// Mitsubishi GX Works2 project: BookEX6_7 Time   PLC: Q13UDV

// global labels: Global
VAR_GLOBAL
  bVar0 AT M5000 : BOOL;
  abArray0 AT M5010 : ARRAY [0..49] OF BOOL;
  sStr0 AT D5000 : STRING[199];
  sStr1 AT D5100 : STRING[199];
  sStr2 AT D5200 : STRING[199];
  sStr3 AT D5300 : STRING[199];
  sStr4 AT D5400 : STRING[199];
  sStr5 AT D5500 : STRING[199];
  sStr6 AT D5600 : STRING[199];
  sStr7 AT D5700 : STRING[199];
  sStr8 AT D5800 : STRING[199];
  sStr9 AT D5900 : STRING[199];
  iVar0 AT D4500 : INT;
  iVar1 AT D4501 : INT;
  iVar2 AT D4502 : INT;
  iVar3 AT D4503 : INT;
  iVar4 AT D4504 : INT;
  iVar5 AT D4505 : INT;
  iVar6 AT D4506 : INT;
  iVar7 AT D4507 : INT;
  iVar8 AT D4508 : INT;
  iVar9 AT D4509 : INT;
  dVar0 AT D4510 : DINT;
  dVar1 AT D4512 : DINT;
  dVar2 AT D4514 : DINT;
  dVar3 AT D4516 : DINT;
  dVar4 AT D4518 : DINT;
  dVar5 AT D4520 : DINT;
  dVar6 AT D4522 : DINT;
  dVar7 AT D4524 : DINT;
  dVar8 AT D4526 : DINT;
  dVar9 AT D4528 : DINT;
  wVar0 AT D4530 : WORD;
  wVar1 AT D4531 : WORD;
  wVar2 AT D4532 : WORD;
  wVar3 AT D4533 : WORD;
  wVar4 AT D4534 : WORD;
  wVar5 AT D4535 : WORD;
  wVar6 AT D4536 : WORD;
  wVar7 AT D4537 : WORD;
  wVar8 AT D4538 : WORD;
  wVar9 AT D4539 : WORD;
  dwVar0 AT D4540 : DWORD;
  dwVar1 AT D4542 : DWORD;
  dwVar2 AT D4544 : DWORD;
  dwVar3 AT D4546 : DWORD;
  dwVar4 AT D4548 : DWORD;
  dwVar5 AT D4550 : DWORD;
  dwVar6 AT D4552 : DWORD;
  dwVar7 AT D4554 : DWORD;
  dwVar8 AT D4556 : DWORD;
  dwVar9 AT D4558 : DWORD;
  fsVar0 AT D4560 : REAL;
  fsVar1 AT D4562 : REAL;
  fsVar2 AT D4564 : REAL;
  fsVar3 AT D4566 : REAL;
  fsVar4 AT D4568 : REAL;
  fsVar5 AT D4570 : REAL;
  fsVar6 AT D4572 : REAL;
  fsVar7 AT D4574 : REAL;
  fsVar8 AT D4576 : REAL;
  fsVar9 AT D4578 : REAL;
  fdVar0 AT D4580 : LREAL;
  tTime0 AT D4620 : TIME;
  tTime1 AT D4622 : TIME;
  tTime2 AT D4624 : TIME;
  tTime3 AT D4626 : TIME;
  tTime4 AT D4628 : TIME;
  tTime5 AT D4630 : TIME;
  tTime6 AT D4632 : TIME;
  tTime7 AT D4634 : TIME;
  tTime8 AT D4636 : TIME;
  tTime9 AT D4638 : TIME;
  tTime10 AT D4640 : TIME;
  bVar1 AT M5001 : BOOL;
  bVar2 AT M5002 : BOOL;
  bVar3 AT M5003 : BOOL;
  bVar4 AT M5004 : BOOL;
  bVar5 AT M5005 : BOOL;
  bVar6 AT M5006 : BOOL;
  bVar7 AT M5007 : BOOL;
  bVar8 AT M5008 : BOOL;
  bVar9 AT M5009 : BOOL;
  abArray1 AT M5060 : ARRAY [0..49] OF BOOL;
  abArray2 AT M5110 : ARRAY [0..49] OF BOOL;
  abArray3 AT M5160 : ARRAY [0..49] OF BOOL;
  abArray4 AT M5210 : ARRAY [0..49] OF BOOL;
  abArray5 AT M5260 : ARRAY [0..49] OF BOOL;
  abArray6 AT M5310 : ARRAY [0..49] OF BOOL;
  abArray7 AT M5360 : ARRAY [0..49] OF BOOL;
  abArray8 AT M5410 : ARRAY [0..49] OF BOOL;
  abArray9 AT M5460 : ARRAY [0..49] OF BOOL;
  fdVar1 AT D4584 : LREAL;
  fdVar2 AT D4588 : LREAL;
  fdVar3 AT D4592 : LREAL;
  fdVar4 AT D4596 : LREAL;
  fdVar5 AT D4600 : LREAL;
  fdVar6 AT D4604 : LREAL;
  fdVar7 AT D4608 : LREAL;
  fdVar8 AT D4612 : LREAL;
  fdVar9 AT D4616 : LREAL;
END_VAR
// user libraries (not included): HMI

FUNCTION ABS_TIME
VAR_INPUT
  t_IN1 : TIME;
  t_IN2 : TIME;
END_VAR
VAR
  tTemp : TIME;
END_VAR
;
tTemp := SUB_TIME(t_IN1, t_IN2);
IF tTemp < T#0ms THEN
	tTemp := MUL_TIME(tTemp, -1);
END_IF;
ABS_TIME := tTemp;
END_FUNCTION

FUNCTION Day2Time
VAR_INPUT
  fs_IN : REAL;
END_VAR
;
Day2Time := DINT_TO_TIME(REAL_TO_DINT(fs_IN * 86400000.0));
END_FUNCTION

FUNCTION fsDIV_TIME
VAR_INPUT
  t_IN1 : TIME;
  fs_IN2 : REAL;
END_VAR
VAR
  dTemp : DINT;
  fsTemp : REAL;
END_VAR
;
dTemp := TIME_TO_DINT(t_IN1);
fsTemp := DINT_TO_REAL(dTemp) / fs_IN2;
fsDIV_TIME := DINT_TO_TIME(REAL_TO_DINT(fsTemp));
END_FUNCTION

FUNCTION fsMUL_TIME
VAR_INPUT
  t_IN1 : TIME;
  fs_IN2 : REAL;
END_VAR
VAR
  dTemp : DINT;
  fsTemp : REAL;
END_VAR
;
dTemp := TIME_TO_DINT(t_IN1);
fsTemp := DINT_TO_REAL(dTemp) * fs_IN2;
fsMUL_TIME := DINT_TO_TIME(REAL_TO_DINT(fsTemp));
END_FUNCTION

FUNCTION Hour2Time
VAR_INPUT
  fs_IN : REAL;
END_VAR
;
Hour2Time := DINT_TO_TIME(REAL_TO_DINT(fs_IN * 3600000.0));
END_FUNCTION

FUNCTION Min2Time
VAR_INPUT
  fs_IN : REAL;
END_VAR
;
Min2Time := DINT_TO_TIME(REAL_TO_DINT(fs_IN * 60000.0));
END_FUNCTION

FUNCTION Sec2Time
VAR_INPUT
  fs_IN : REAL;
END_VAR
;
Sec2Time := DINT_TO_TIME(REAL_TO_DINT(fs_IN * 1000.0));
END_FUNCTION

PROGRAM ExADDTIME
(* structured ladder/FBD written out as ST: instructions are called as NAME(EN, inputs, outputs); _pN, _eN, _tN stand for wires *)
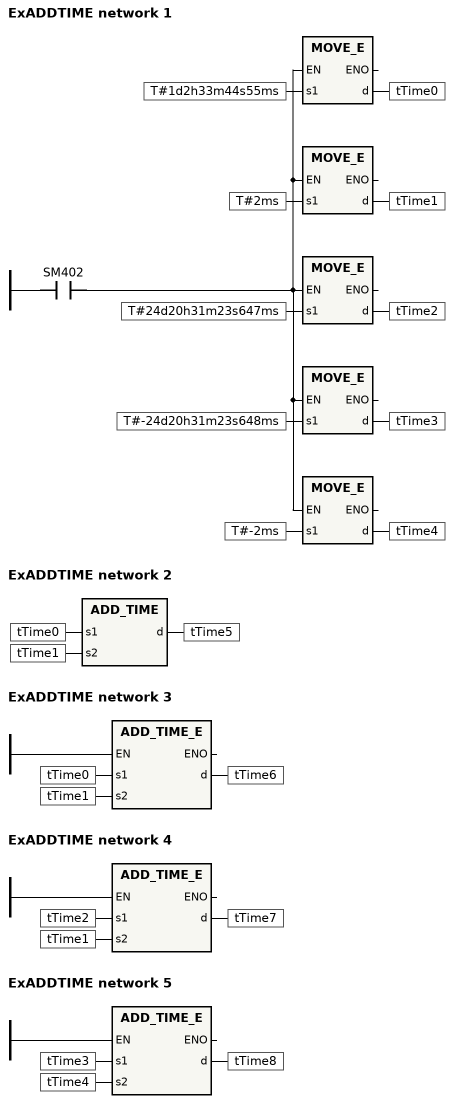
(* network 1 *)
MOVE_E(SM402, T#1d2h33m44s55ms, tTime0);
MOVE_E(SM402, T#2ms, tTime1);
MOVE_E(SM402, T#24d20h31m23s647ms, tTime2);
MOVE_E(SM402, T#-24d20h31m23s648ms, tTime3);
MOVE_E(SM402, T#-2ms, tTime4);
(* network 2 *)
tTime5 := ADD_TIME(tTime0, tTime1);
(* network 3 *)
ADD_TIME_E(TRUE, tTime0, tTime1, tTime6);
(* network 4 *)
ADD_TIME_E(TRUE, tTime2, tTime1, tTime7);
(* network 5 *)
ADD_TIME_E(TRUE, tTime3, tTime4, tTime8);
END_PROGRAM

PROGRAM ExDIVTIME
VAR
  tTime20 : TIME;
  tTime21 : TIME;
  tTime22 : TIME;
  tTime23 : TIME;
  tTime24 : TIME;
  tTime25 : TIME;
  tTime26 : TIME;
  tTime27 : TIME;
  tTime28 : TIME;
  tTime29 : TIME;
END_VAR
(* structured ladder/FBD written out as ST: instructions are called as NAME(EN, inputs, outputs); _pN, _eN, _tN stand for wires *)
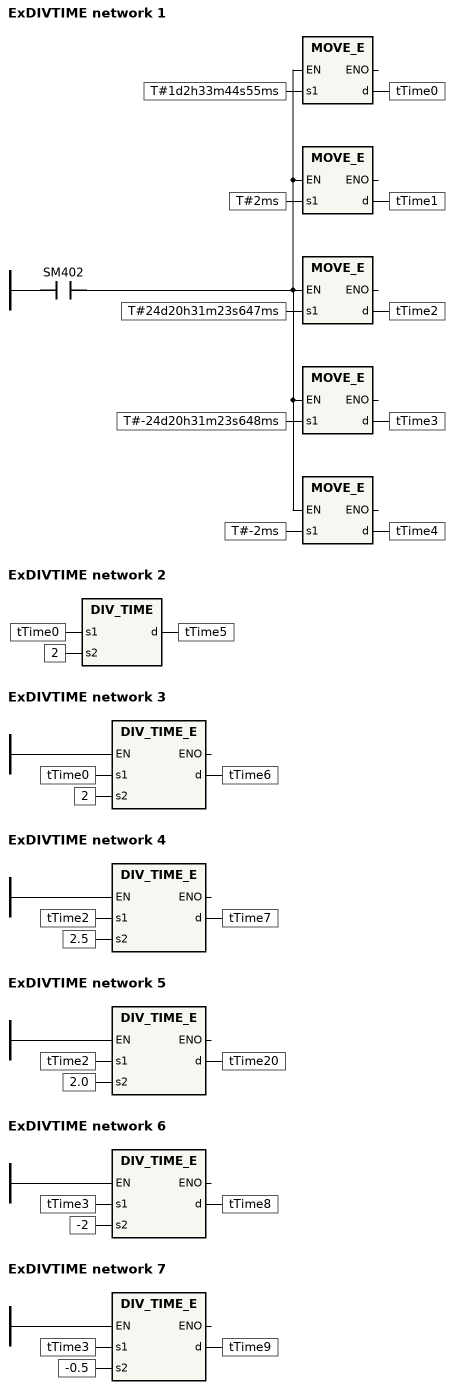
(* network 1 *)
MOVE_E(SM402, T#1d2h33m44s55ms, tTime0);
MOVE_E(SM402, T#2ms, tTime1);
MOVE_E(SM402, T#24d20h31m23s647ms, tTime2);
MOVE_E(SM402, T#-24d20h31m23s648ms, tTime3);
MOVE_E(SM402, T#-2ms, tTime4);
(* network 2 *)
tTime5 := DIV_TIME(tTime0, 2);
(* network 3 *)
DIV_TIME_E(TRUE, tTime0, 2, tTime6);
(* network 4 *)
DIV_TIME_E(TRUE, tTime2, 2.5, tTime7);
(* network 5 *)
DIV_TIME_E(TRUE, tTime2, 2.0, tTime20);
(* network 6 *)
DIV_TIME_E(TRUE, tTime3, -2, tTime8);
(* network 7 *)
DIV_TIME_E(TRUE, tTime3, -0.5, tTime9);
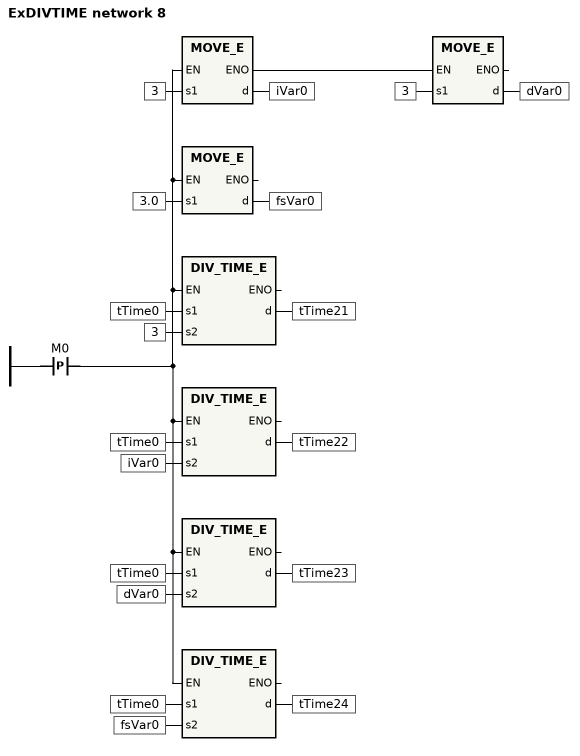
(* network 8 *)
_p1 := LDP(TRUE, M0);
_e2 := MOVE_E(_p1, 3, iVar0);
MOVE_E(_e2, 3, dVar0);
MOVE_E(_p1, 3.0, fsVar0);
DIV_TIME_E(_p1, tTime0, 3, tTime21);
DIV_TIME_E(_p1, tTime0, iVar0, tTime22);
DIV_TIME_E(_p1, tTime0, dVar0, tTime23);
DIV_TIME_E(_p1, tTime0, fsVar0, tTime24);
END_PROGRAM

PROGRAM ExFB
(* structured ladder/FBD written out as ST: instructions are called as NAME(EN, inputs, outputs); _pN, _eN, _tN stand for wires *)
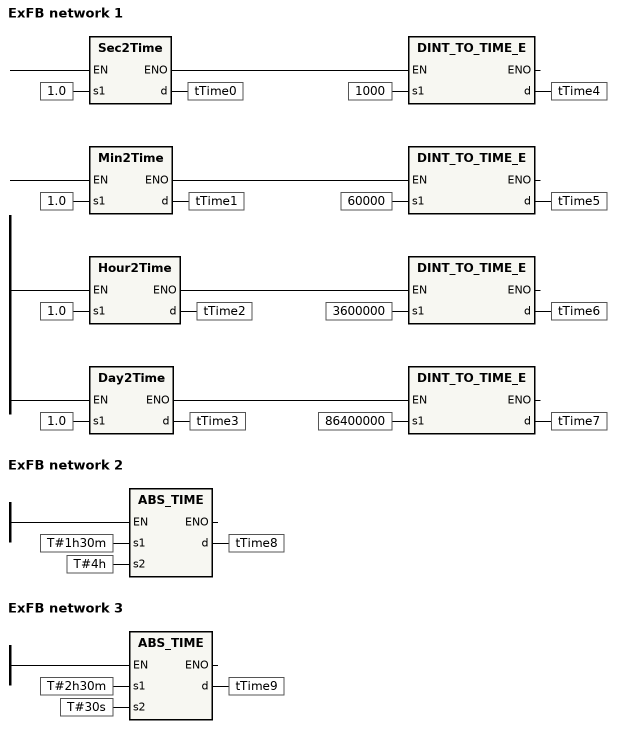
(* network 1 *)
_e1 := Sec2Time(TRUE, 1.0, tTime0);
DINT_TO_TIME_E(_e1, 1000, tTime4);
_e2 := Min2Time(TRUE, 1.0, tTime1);
DINT_TO_TIME_E(_e2, 60000, tTime5);
_e3 := Hour2Time(TRUE, 1.0, tTime2);
DINT_TO_TIME_E(_e3, 3600000, tTime6);
_e4 := Day2Time(TRUE, 1.0, tTime3);
DINT_TO_TIME_E(_e4, 86400000, tTime7);
(* network 2 *)
ABS_TIME(TRUE, T#1h30m, T#4h, tTime8);
(* network 3 *)
ABS_TIME(TRUE, T#2h30m, T#30s, tTime9);
END_PROGRAM

PROGRAM ExMUL_DIV
VAR
  tTime20 : TIME;
  tTime21 : TIME;
  tTime22 : TIME;
  tTime23 : TIME;
  tTime24 : TIME;
  tTime25 : TIME;
  tTime26 : TIME;
  tTime27 : TIME;
  tTime28 : TIME;
  tTime29 : TIME;
  tTime30 : TIME;
  tTime31 : TIME;
  tTime32 : TIME;
  tTime33 : TIME;
  tTime34 : TIME;
  tTime35 : TIME;
  tTime36 : TIME;
  tTime37 : TIME;
  tTime38 : TIME;
  tTime39 : TIME;
  tTime40 : TIME;
END_VAR
(* structured ladder/FBD written out as ST: instructions are called as NAME(EN, inputs, outputs); _pN, _eN, _tN stand for wires *)
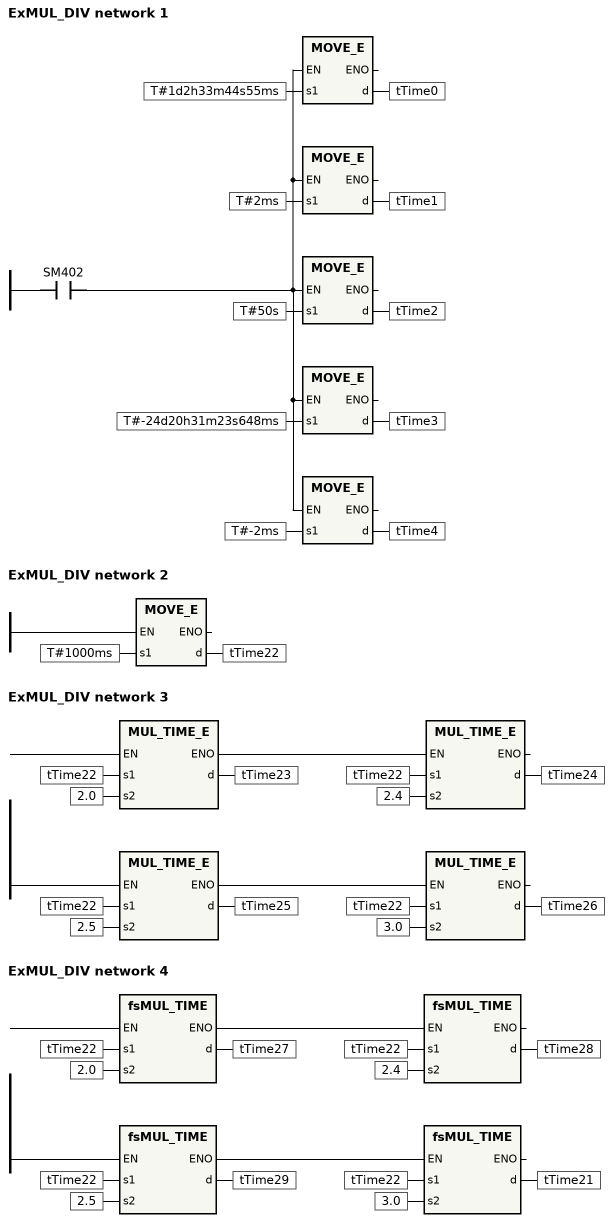
(* network 1 *)
MOVE_E(SM402, T#1d2h33m44s55ms, tTime0);
MOVE_E(SM402, T#2ms, tTime1);
MOVE_E(SM402, T#50s, tTime2);
MOVE_E(SM402, T#-24d20h31m23s648ms, tTime3);
MOVE_E(SM402, T#-2ms, tTime4);
(* network 2 *)
MOVE_E(TRUE, T#1000ms, tTime22);
(* network 3 *)
_e1 := MUL_TIME_E(TRUE, tTime22, 2.0, tTime23);
MUL_TIME_E(_e1, tTime22, 2.4, tTime24);
_e2 := MUL_TIME_E(TRUE, tTime22, 2.5, tTime25);
MUL_TIME_E(_e2, tTime22, 3.0, tTime26);
(* network 4 *)
_e1 := fsMUL_TIME(TRUE, tTime22, 2.0, tTime27);
fsMUL_TIME(_e1, tTime22, 2.4, tTime28);
_e2 := fsMUL_TIME(TRUE, tTime22, 2.5, tTime29);
fsMUL_TIME(_e2, tTime22, 3.0, tTime21);
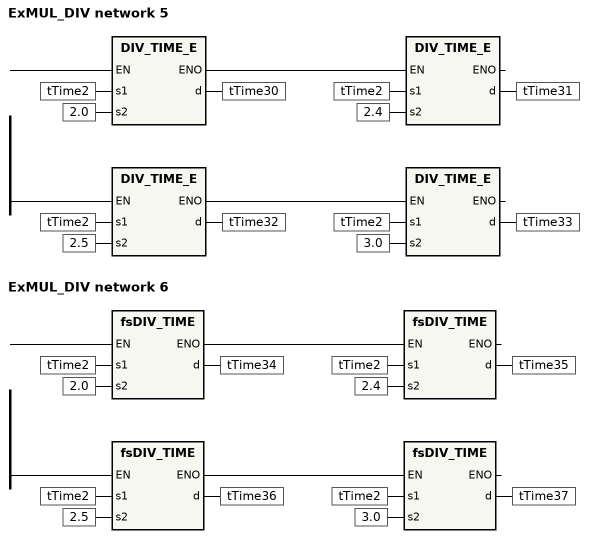
(* network 5 *)
_e1 := DIV_TIME_E(TRUE, tTime2, 2.0, tTime30);
DIV_TIME_E(_e1, tTime2, 2.4, tTime31);
_e2 := DIV_TIME_E(TRUE, tTime2, 2.5, tTime32);
DIV_TIME_E(_e2, tTime2, 3.0, tTime33);
(* network 6 *)
_e1 := fsDIV_TIME(TRUE, tTime2, 2.0, tTime34);
fsDIV_TIME(_e1, tTime2, 2.4, tTime35);
_e2 := fsDIV_TIME(TRUE, tTime2, 2.5, tTime36);
fsDIV_TIME(_e2, tTime2, 3.0, tTime37);
END_PROGRAM

PROGRAM ExMULTIME
(* structured ladder/FBD written out as ST: instructions are called as NAME(EN, inputs, outputs); _pN, _eN, _tN stand for wires *)
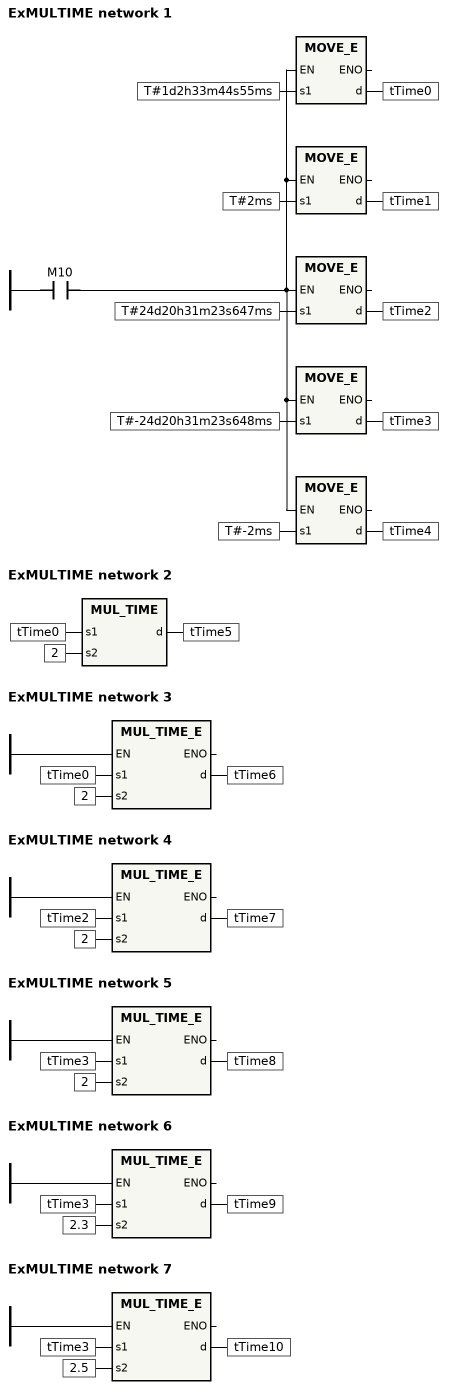
(* network 1 *)
MOVE_E(M10, T#1d2h33m44s55ms, tTime0);
MOVE_E(M10, T#2ms, tTime1);
MOVE_E(M10, T#24d20h31m23s647ms, tTime2);
MOVE_E(M10, T#-24d20h31m23s648ms, tTime3);
MOVE_E(M10, T#-2ms, tTime4);
(* network 2 *)
tTime5 := MUL_TIME(tTime0, 2);
(* network 3 *)
MUL_TIME_E(TRUE, tTime0, 2, tTime6);
(* network 4 *)
MUL_TIME_E(TRUE, tTime2, 2, tTime7);
(* network 5 *)
MUL_TIME_E(TRUE, tTime3, 2, tTime8);
(* network 6 *)
MUL_TIME_E(TRUE, tTime3, 2.3, tTime9);
(* network 7 *)
MUL_TIME_E(TRUE, tTime3, 2.5, tTime10);
END_PROGRAM

PROGRAM ExSUBTIME
(* structured ladder/FBD written out as ST: instructions are called as NAME(EN, inputs, outputs); _pN, _eN, _tN stand for wires *)
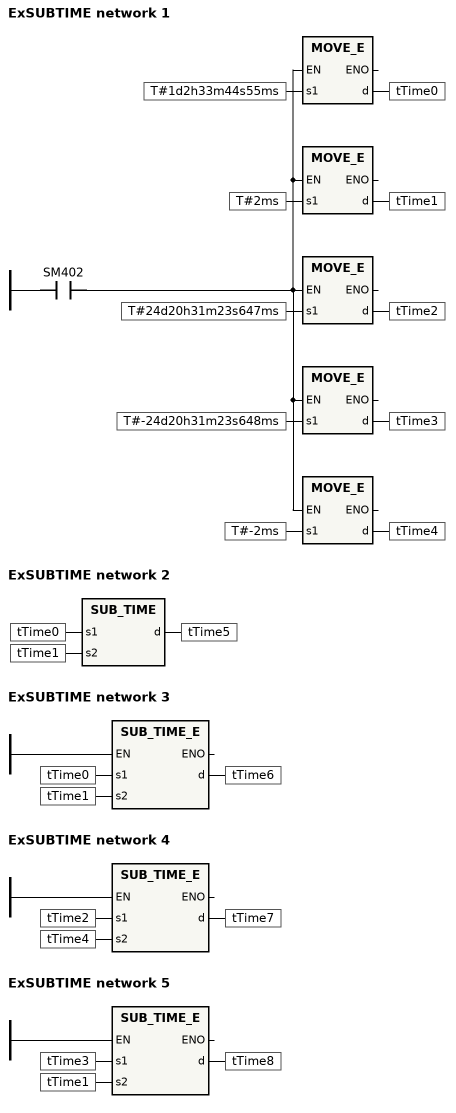
(* network 1 *)
MOVE_E(SM402, T#1d2h33m44s55ms, tTime0);
MOVE_E(SM402, T#2ms, tTime1);
MOVE_E(SM402, T#24d20h31m23s647ms, tTime2);
MOVE_E(SM402, T#-24d20h31m23s648ms, tTime3);
MOVE_E(SM402, T#-2ms, tTime4);
(* network 2 *)
tTime5 := SUB_TIME(tTime0, tTime1);
(* network 3 *)
SUB_TIME_E(TRUE, tTime0, tTime1, tTime6);
(* network 4 *)
SUB_TIME_E(TRUE, tTime2, tTime4, tTime7);
(* network 5 *)
SUB_TIME_E(TRUE, tTime3, tTime1, tTime8);
END_PROGRAM

PROGRAM stt
;
tTime2 := ADD_TIME( tTime0 , tTime1 );
bVar0 := ADD_TIME_E( TRUE,  tTime0 , tTime1, tTime2 );
tTime2 := SUB_TIME( tTime0 , tTime1 );
END_PROGRAM

PROGRAM ExDIV_ST
VAR
  tTime20 : TIME;
  tTime21 : TIME;
  tTime22 : TIME;
  tTime23 : TIME;
  tTime24 : TIME;
  tTime25 : TIME;
  tTime26 : TIME;
  tTime27 : TIME;
  tTime28 : TIME;
  tTime29 : TIME;
  tTime30 : TIME;
  tTime31 : TIME;
  tTime32 : TIME;
  tTime33 : TIME;
  tTime34 : TIME;
  tTime35 : TIME;
  tTime36 : TIME;
  tTime37 : TIME;
  tTime38 : TIME;
  tTime39 : TIME;
END_VAR
;
iVar1 := 3;
dVar1 := 3;
fsVar1 := 3.0;
tTime0 := T#1d2h33m44s55ms;
 
tTime29 := tTime0 + tTime1;
tTime28 := tTime0 - tTime1;

tTime31 := tTime0 * 3;
tTime32 := tTime0 * iVar1;
tTime33 := tTime0 * dVar1;
tTime34 := tTime0 * fsVar1;
tTime35 := MUL_TIME(tTime0, fsVar1);

tTime21 := tTime0 / 3;
tTime22 := tTime0 / iVar1;
tTime23 := tTime0 / dVar1;
tTime24 := tTime0 / fsVar1;
tTime25 := DIV_TIME(tTime0, fsVar1);

(*
tTime34 := tTime0 * fsVar1;
tTime35 := MUL_TIME(tTime0, fsVar1);
tTime24 := tTime0 / fsVar1;
tTime25 := DIV_TIME(tTime0, fsVar1);
*)
END_PROGRAM
